// TIA Portal V17 export
// export: Created 2024-09-02T12:50:18.3911092Z, ExportSetting WithDefaults, DisplayName Totally Integrated Automation Portal, DisplayVersion V17, DisplayName TIA Portal Openness, DisplayVersion V17, DisplayName TIA Portal Version Control Interface, DisplayVersion V17, DisplayName STEP 7 Professional, DisplayVersion V17, DisplayName STEP 7 Safety, DisplayVersion V17, DisplayName WinCC Professional, DisplayVersion V17
DATA_BLOCK "LTLL_DeviceDiag_OP70"   // DB583
TITLE = LTLL_DeviceDiag
{ S7_Optimized_Access := 'TRUE'; DB_Accessible_From_OPC_UA := 'FALSE' }
AUTHOR : Siemens
FAMILY : HMI_Lite
NAME : LTLL_DeviceDiag
VERSION : 8.10
// stored: AutoNumber true, DBAccessibleFromOPCUA false, InstanceOfName LTLL_typeDeviceDiag, InstanceOfType UDT, IsOnlyStoredInLoadMemory false, IsWriteProtectedInAS false
"LTLL_typeDeviceDiag"
   // VAR
   //    "version" { S7_SetPoint := 'True'} : "LTLL_typeVersion";
   //    screenRFID : Struct
   //       selectedDevice : UInt;
   //       done : Bool;
   //       busy : Bool;
   //       warning : Bool;
   //       error : Bool;
   //       status : DWord;
   //       statusIDForText : DWord;
   //       transponderPresence : Bool;
   //       transponderPresenceChanged : Bool;
   //       iidCmdStruct { S7_SetPoint := 'True'} : IID_CMD_STRUCT;
   //    END_STRUCT;
   //    screenSinamics : Struct
   //       selectedDriveobject : Byte;
   //       driveobjectType : Byte;
   //       controlWord : Word;
   //       statusWord : Word;
   //       posStatusWord : Word;
   //       posSetValue : DInt;
   //       posActValue : DInt;
   //       speedActValue : DInt;
   //       override : Real;
   //       blockSelect : Int;
   //       blockCurrent : DInt;
   //       faultCode : Array[0..7] of Word;
   //       alarmCode : Array[0..3] of Word;
   //       dimension : Word;
   //       freqSetValueDword : DWord;
   //       freqSetValue : Real;
   //       freqActValueDword : DWord;
   //       freqActValue : Real;
   //       safetyStatusWord : Word;
   //       error : Bool;
   //    END_STRUCT;
   //    screenMotorstarter : Struct
   //       selectedObject : USInt;
   //       selectedDeviceType : Byte;
   //       controlStatusProtection : Struct
   //          control : Struct
   //             motorRight : Bool;
   //             motorLeft : Bool;
   //             anlaufAktiv : Bool;
   //             auslaufAktiv : Bool;
   //             notstartAktiv : Bool;
   //             bremsausgangAktiv : Bool;
   //          END_STRUCT;
   //          protection : Struct
   //             ueberlastAbschaltung : Bool;
   //             thermischesMotormodellUeberlast : Bool;
   //             schaltelementUeberlast : Bool;
   //             schaltelementDefekt : Bool;
   //             abkuehlzeitAktiv : Bool;
   //             motorBlockierung : Bool;
   //          END_STRUCT;
   //          status : Struct
   //             bereit : Bool;
   //             motorEin : Bool;
   //             sammelfehler : Bool;
   //             sammelwarnung : Bool;
   //             versorgElekToLow : Bool;
   //             versorgSchaltelementFehlt : Bool;
   //             nullstromAbschaltung : Bool;
   //             unsymmetrie : Bool;
   //             verriegelungszeitAktiv : Bool;
   //             eingang1 : Bool;
   //             eingang2 : Bool;
   //             eingang3 : Bool;
   //             eingang4 : Bool;
   //          END_STRUCT;
   //       END_STRUCT;
   //       dataStatistics : Struct
   //          data : Struct
   //             phaseCurrent1 : LReal;
   //             phaseCurrent2 : LReal;
   //             phaseCurrent3 : LReal;
   //             motorWaermung : Word;
   //             unbalance : Bool;
   //             valueUnbalance : Byte;
   //          END_STRUCT;
   //          statistics : Struct
   //             operatingHourDevice : UDInt;
   //             operatingHourMotor : UDInt;
   //             countMotorStartRight : UDInt;
   //             countMotorStartLeft : UDInt;
   //             motorCurrent : LReal;
   //             lastTrippingCurrent : LReal;
   //             countMotorOverloadRelease : UInt;
   //             countSwitchElementOverloadRelease : UInt;
   //          END_STRUCT;
   //       END_STRUCT;
   //       logbook : Struct
   //          deviceErrors { S7_SetPoint := 'True'} : Array[0..20] of "LTLL_typeMotorStarterLogbook";
   //          trippingOperations { S7_SetPoint := 'True'} : Array[0..20] of "LTLL_typeMotorStarterLogbook";
   //          events { S7_SetPoint := 'True'} : Array[0..20] of "LTLL_typeMotorStarterLogbook";
   //       END_STRUCT;
   //    END_STRUCT;
   // END_VAR
BEGIN
   "version".high := 16#08;
   "version".middle := 16#01;
   "version".low := 16#00;
END_DATA_BLOCK
